// TIA Portal project "Safety f-cpu" (V17)

(* hardware
DEVICE "S7-1200 station_1"  S7-1200 Station
   slot 0: "Rack_0"  S7-1200 Rack  Rack  V1.0
   slot 1: "PLC_1"  CPU 1214FC DC/DC/DC  6ES7 214-1AF40-0XB0  V4.5
*)

// ===== PLC "PLC_1"  CPU 1214FC DC/DC/DC =====

VAR_GLOBAL   // PLC tag table "Default tag table"
   "E_Stop" AT %I0.0 : Bool;
   "Safe_Output" AT %Q0.0 : Bool;
   "Gate_Closed" AT %I0.3 : Bool;
   "Fault" AT %I0.4 : Bool;
   "Safety_Ok" AT %Q0.1 : Bool;
   "Reset_Pressed" AT %I0.6 : Bool;
   "Reset_Latch" AT %Q0.2 : Bool;
END_VAR

DATA_BLOCK "Main_Safety_RTG1_DB"   // DB1, F_DB
{ S7_Optimized_Access := 'TRUE' }
NAME : FUSI
VERSION : 0.1
// stored: InstanceOfName Main_Safety_RTG1
"Main_Safety_RTG1"
BEGIN
END_DATA_BLOCK

FUNCTION_BLOCK "Main_Safety_RTG1"   // FB1, F_FBD
{ S7_Optimized_Access := 'TRUE' }
BEGIN
END_FUNCTION_BLOCK

FUNCTION "Safety_Logic" : Void   // FC1, LAD
{ S7_Optimized_Access := 'TRUE' }
VERSION : 0.1
BEGIN

REGION Network 1
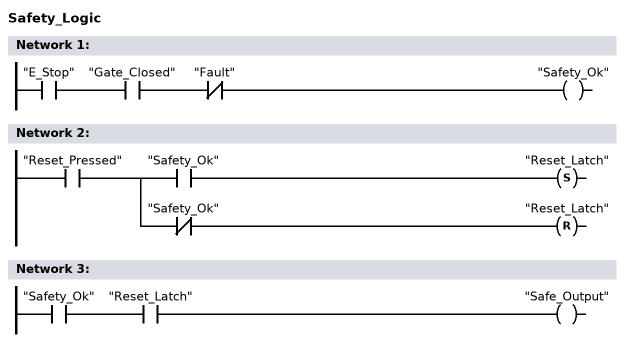
   RUNG wire#powerrail
      Contact( "E_Stop" )
      Contact( "Gate_Closed" )
      I_Contact( "Fault" )
      Coil( "Safety_Ok" )
   END_RUNG
   // the same network as SCL:
   "Safety_Ok" := "E_Stop" AND "Gate_Closed" AND NOT "Fault";
END_REGION

REGION Network 2
   RUNG wire#powerrail
      Contact( "Reset_Pressed" )
      wire#w1
      Contact( "Safety_Ok" )
      S_Coil( "Reset_Latch" )
   END_RUNG
   RUNG wire#w1
      I_Contact( "Safety_Ok" )
      R_Coil( "Reset_Latch" )
   END_RUNG
   // the same network as SCL:
   IF "Reset_Pressed" AND "Safety_Ok" THEN "Reset_Latch" := TRUE; END_IF;
   IF "Reset_Pressed" AND NOT "Safety_Ok" THEN "Reset_Latch" := FALSE; END_IF;
END_REGION

REGION Network 3
   RUNG wire#powerrail
      Contact( "Safety_Ok" )
      Contact( "Reset_Latch" )
      Coil( "Safe_Output" )
   END_RUNG
   // the same network as SCL:
   "Safe_Output" := "Safety_Ok" AND "Reset_Latch";
END_REGION
END_FUNCTION

ORGANIZATION_BLOCK "Main"   // OB1, LAD, ProgramCycle
TITLE = "Main Program Sweep (Cycle)"
{ S7_Optimized_Access := 'TRUE' }
VERSION : 0.1
   VAR_INPUT
      Initial_Call : Bool;   // Initial call of this OB
      Remanence : Bool;   // =True, if remanent data are available
   END_VAR
BEGIN

REGION Network 1
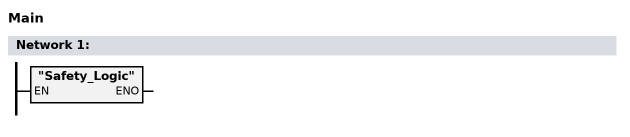
   RUNG wire#powerrail
      "Safety_Logic"()
   END_RUNG
   // the same network as SCL:
   "Safety_Logic"();
END_REGION
END_ORGANIZATION_BLOCK